// TIA Portal V17 export
FUNCTION "FC_Name" : Void   // FC, LAD
{ S7_Optimized_Access := 'TRUE' }
// stored: AutoNumber true
BEGIN
END_FUNCTION
